Staubli VAL3: sendData.pgx

program sendData(sio& x_UdpSocket, num& x_nData[], bool& x_bError)
begin

    if (size(x_nData) == 0)
      x_bError = true
      logMsg("ros2_server::sendUdpData : empty buffer!", 3)
      return
    endIf

    if(sioSet(x_UdpSocket, x_nData) != size(x_nData))
      logMsg("ros2_server::sendUdpData : failed to write all bytes to socket", 3)
      x_bError = true
    else
      x_bError = false
    endIf

end
